TYPE ST_OutputsLiftTable :
STRUCT
	HW 							: ST_HW_OutputsLiftTable; //Hardware outputs
	LiftTableEnableTransport	: BOOL; //Enable transport when lift is done
END_STRUCT
END_TYPE

(* stored: Version 1.1.0.1, ProductVersion 3.1.4024.9
   DUT ST_OutputsLiftTable: Id {e6597d17-e055-4d79-898f-c4e481c72b73} *)
